KUKA KRL program: braketestpark.src, braketestpark.dat

--- braketestpark.src ---
&ACCESS RVP2
&REL 3
&COMMENT parkposition
&PARAM DISKPATH = KRC:\R1\TP\BrakeTest
&PARAM TEMPLATE = C:\KRC\Roboter\Template\vorgabe
&PARAM EDITMASK = *
DEF BrakeTestPark( )
;FOLD INI
  ;FOLD BASISTECH INI
    GLOBAL INTERRUPT DECL 3 WHEN $STOPMESS==TRUE DO IR_STOPM ( )
    INTERRUPT ON 3
    BAS (#INITMOV,0 )
  ;ENDFOLD (BASISTECH INI)
;FOLD GRIPPERTECH INI
USER_GRP(0,DUMMY,DUMMY,GDEFAULT)
;ENDFOLD (GRIPPERTECH INI)
  ;FOLD USER INI
    ;Make your modifications here

  ;ENDFOLD (USER INI)
;ENDFOLD (INI)

;Teach here the motion to the parking position. The parking position is needed when the robot has failed the brake test.
;FOLD PTP Parkposition  Vel= 10 % DEFAULT;%{PE}%R 5.4.24,%MKUKATPBASIS,%CMOVE,%VPTP,%P 1:PTP, 2:Parkposition, 3:, 5:10, 7:DEFAULT
$BWDSTART = FALSE
PDAT_ACT=PDEFAULT
FDAT_ACT=FParkposition
BAS(#PTP_PARAMS,10)
PTP XParkposition
;ENDFOLD

END

--- braketestpark.dat ---
&ACCESS RVP2
&REL 3
&COMMENT parkposition
&PARAM DISKPATH = KRC:\R1\TP\BrakeTest
&PARAM TEMPLATE = C:\KRC\Roboter\Template\vorgabe
&PARAM EDITMASK = *
DEFDAT  braketestpark PUBLIC
;FOLD EXTERNAL DECLARATIONS;%{PE}%MKUKATPBASIS,%CEXT,%VCOMMON,%P
;FOLD GRIPPERTECH EXT
EXT  H50 (INT  :IN,INT  :IN,INT  :IN,GRP_TYP  :IN )
;ENDFOLD (GRIPPERTECH EXT)
;FOLD SPOTTECH EXT
EXT  USERSPOT (S_COMMAND  :IN,SPOT_TYPE  :IN )
;ENDFOLD (SPOTTECH EXT)
;FOLD BASISTECH EXT;%{PE}%MKUKATPBASIS,%CEXT,%VEXT,%P
EXT  BAS (BAS_COMMAND  :IN,REAL  :IN )
DECL INT SUCCESS
;ENDFOLD (BASISTECH EXT)
;FOLD USER EXT;%{E}%MKUKATPUSER,%CEXT,%VEXT,%P
;Make here your modifications

;ENDFOLD (USER EXT)
;ENDFOLD (EXTERNAL DECLERATIONS)
DECL BASIS_SUGG_T LAST_BASIS={POINT1[] "P0                      ",POINT2[] "P0                      ",CP_PARAMS[] "CPDAT0                  ",PTP_PARAMS[] "PDAT0                   ",CONT[] "                        ",CP_VEL[] "2.0                     ",PTP_VEL[] "100                     ",SPL_NAME[] "S0                      "}
DECL E6AXIS xParkposition={A1 -120.744003,A2 -100.945297,A3 80.7224731,A4 -10.1595001,A5 70.2619934,A6 120.210899,E1 1001.177,E2 0.0,E3 0.0,E4 0.0,E5 0.0,E6 0.0}
DECL FDAT FParkposition={TOOL_NO 0,BASE_NO 0,IPO_FRAME #BASE,POINT2[] " "}
ENDDAT
